(*
SPDX-FileCopyrightText: c 2026 Oleksandr Tiutyk <trofimich@gmail.com>
SPDX-License-Identifier: MIT
License: https://opensource.org/license/mit
*)

(*!
<summary>Groups the three raw representations tested by the range converter suite.</summary>
<description>
Owns persistent child storage and fixed parent associations. Use in one task without reentry and do not copy the group.
Children is borrowed and must not be modified by application code. Constructor callbacks are not used.
</description>
*)

{attribute 'no_assign'}
{attribute 'no_explicit_call' := 'do not call this function block directly'}
FUNCTION_BLOCK RangeAnalogValueConverterTest EXTENDS TOF_Testing.TestGroup<3>
VAR_STAT
	{attribute 'hide'}
	_ClassName : STRING := __POUNAME();
END_VAR
VAR
	_Test16Bit : RangeAnalogValueConverter16BitTest(name := "Test16Bit", parent := THIS^);
	_Test32Bit : RangeAnalogValueConverter32BitTest(name := "Test32Bit", parent := THIS^);
	_Test32Real : RangeAnalogValueConverter32RealTest(name := "Test32Real", parent := THIS^);

	_Children : ARRAY [0.._ChildCount - 1] OF TOF_Testing.ITestElement :=
	[
		_Test16Bit,
		_Test32Bit,
		_Test32Real
	];
END_VAR

//! <summary>Borrows the fixed array of this concrete group; do not modify it.</summary>
{attribute 'monitoring' := 'call'}
PROPERTY Children : REFERENCE TO ARRAY [0.._ChildCount - 1] OF TOF_Testing.ITestElement
GET
Children REF= _Children;
END_GET
END_PROPERTY

//! <summary>Borrows the concrete class name for the lifetime of this instance; callers must not modify it.</summary>
{attribute 'monitoring' := 'call'}
PROPERTY ClassName : REFERENCE TO STRING
GET
ClassName REF= _ClassName;
END_GET
END_PROPERTY

//! <summary>Borrows the compiler-initialized namespace; callers must not modify the returned reference.</summary>
{attribute 'monitoring' := 'call'}
PROPERTY NamespaceName : REFERENCE TO STRING
GET
NamespaceName REF= CurrentNamespace.Name;
END_GET
END_PROPERTY

//! <summary>Reports the complete concrete instance size, excluding separately allocated storage.</summary>
{attribute 'monitoring' := 'call'}
PROPERTY SelfSize : ULINT
GET
SelfSize := XSIZEOF(THIS^);
END_GET
END_PROPERTY

END_FUNCTION_BLOCK

(* stored: Version 1.1.0.1
   POU RangeAnalogValueConverterTest: Id {79b9f598-a289-4b39-880b-c398c6b2163a}, SpecialFunc None
   Property Children: Id {3a70d424-b9aa-43e8-ae82-e6e3b348fcf7}
   Get Get: Id {59c5bb8e-cb9f-4013-ad08-7751882ea92d}
   Property ClassName: Id {8d4d507f-46be-4526-a369-376788bb5a90}
   Get Get: Id {d3e8a331-9150-434e-89fe-51b5432ad77e}
   Property NamespaceName: Id {53d46b4f-752d-4973-98c9-8d9f4b8a93e6}
   Get Get: Id {19582c34-ba89-45dc-a127-2d14f2d0132c}
   Property SelfSize: Id {4e9cb01b-26c4-42f1-ae05-0e7d93b05e42}
   Get Get: Id {17ce538b-fea6-43df-9420-ac9cafcbffab} *)
